FUNCTION_BLOCK RemoveMoverFromGroup  IMPLEMENTS I_Task
VAR
	mcRemoveAxisFromGroup : MC_RemoveAxisFromGroup;
	_caGroup : I_CollisionGroup;
	_Leave: BOOL;
	State: INT;
	_Done: BOOL;
	_Error: BOOL;
	_Busy: BOOL;
	_ErrorId : UDINT;
END_VAR

METHOD Abort : BOOL
mcRemoveAxisFromGroup.Execute := FALSE;
_Leave := FALSE;
Abort := true;
State := 0;
END_METHOD

PROPERTY Busy : BOOL
GET
Busy := _Busy;
END_GET
END_PROPERTY

METHOD Cycle : HRESULT
VAR_INPUT
END_VAR
IF _caGroup = 0 THEN
	Cycle := -1;
	RETURN;
END_IF

_Done := mcRemoveAxisFromGroup.Done OR _Done;
_Error := mcRemoveAxisFromGroup.Error OR _Error;
IF mcRemoveAxisFromGroup.ErrorId <> 0 THEN
	_ErrorId := mcRemoveAxisFromGroup.ErrorId;
END_IF

mcRemoveAxisFromGroup(AxesGroup := _caGroup.GroupRef);
mcRemoveAxisFromGroup.Execute := FALSE;
END_METHOD

PROPERTY Done : BOOL
GET
Done := _Done;
END_GET
END_PROPERTY

PROPERTY Error : BOOL
GET
Error := _Error;
END_GET
END_PROPERTY

METHOD Execute : HRESULT
VAR_INPUT
	AxisID : IDENT_IN_GROUP_REF;
END_VAR
IF mcRemoveAxisFromGroup.Execute THEN
	Execute := -1;
	RETURN;
END_IF

IF _caGroup = 0 THEN
	Execute := -2;
	RETURN;
END_IF

mcRemoveAxisFromGroup.Execute := TRUE;
mcRemoveAxisFromGroup.IdentInGroup := AxisID;
END_METHOD

PROPERTY MyCollisionGroup : I_CollisionGroup
GET
MyCollisionGroup := _caGroup;
END_GET
SET
IF MyCollisionGroup <> 0 THEN
	_caGroup := MyCollisionGroup;
END_IF
END_SET
END_PROPERTY

END_FUNCTION_BLOCK

(* stored: Version 1.1.0.1
   POU RemoveMoverFromGroup: Id {33b40d75-d01d-4ded-8ec6-9cce1233ee05}, SpecialFunc None
   Method Abort: Id {5f143af2-570c-4ae8-a3e1-0058182dca35}
   Property Busy: Id {4c896568-0b71-4fcb-aae9-48e820feba6a}
   Get Get: Id {cfe75508-e331-4ec2-b0e4-6348712fde64}
   Method Cycle: Id {8ab278dc-8dad-4664-bee0-b30bd7e80670}
   Property Done: Id {df5f6adc-b19a-43ee-9c29-ce0366089b3b}
   Get Get: Id {db8fd3e5-af5e-4dfd-92cb-67d05f7143dd}
   Property Error: Id {4c4622ee-476d-4102-9326-d0b4e3863730}
   Get Get: Id {8d4ba5ab-efd2-46bd-9b3f-25a7fea1cc5a}
   Method Execute: Id {efa5d448-3299-4d10-a02c-919548e37d2d}
   Property MyCollisionGroup: Id {f47e6921-e615-4f7a-b716-f9c7b5078fd6}
   Get Get: Id {f0470e42-6eeb-4eb6-90b1-c6a9786719dd}
   Set Set: Id {f1fd62e0-9180-4b79-858e-6bf0b96aa520} *)
